// TIA Portal V20 export
FUNCTION "FC_DataToSafety" : Void   // FC10120, SCL
{ S7_Optimized_Access := 'TRUE' }
// stored: AutoNumber false, SetENOAutomatically false
BEGIN
   REGION Transfert des datas dans le DB Buffer
       "DB_DataToSafety".OpenShutterButton := "DB_McpKeyboardSignals".sRemoteOpenShutter.sKeySWStatus;
       "DB_DataToSafety".ResetEmergencyStop := "MCP1_In".reset;
       "DB_DataToSafety".JOG_Mod := "LBP_ModeGroup".E_JOG;
       "DB_DataToSafety".Activation_Axis := "DB_DigitalOutputs".sAxisActivation.sSWStatus;
       "DB_DataToSafety".CloseShutter := "DB_DataToSafety".CloseShutter;
   END_REGION
END_FUNCTION
